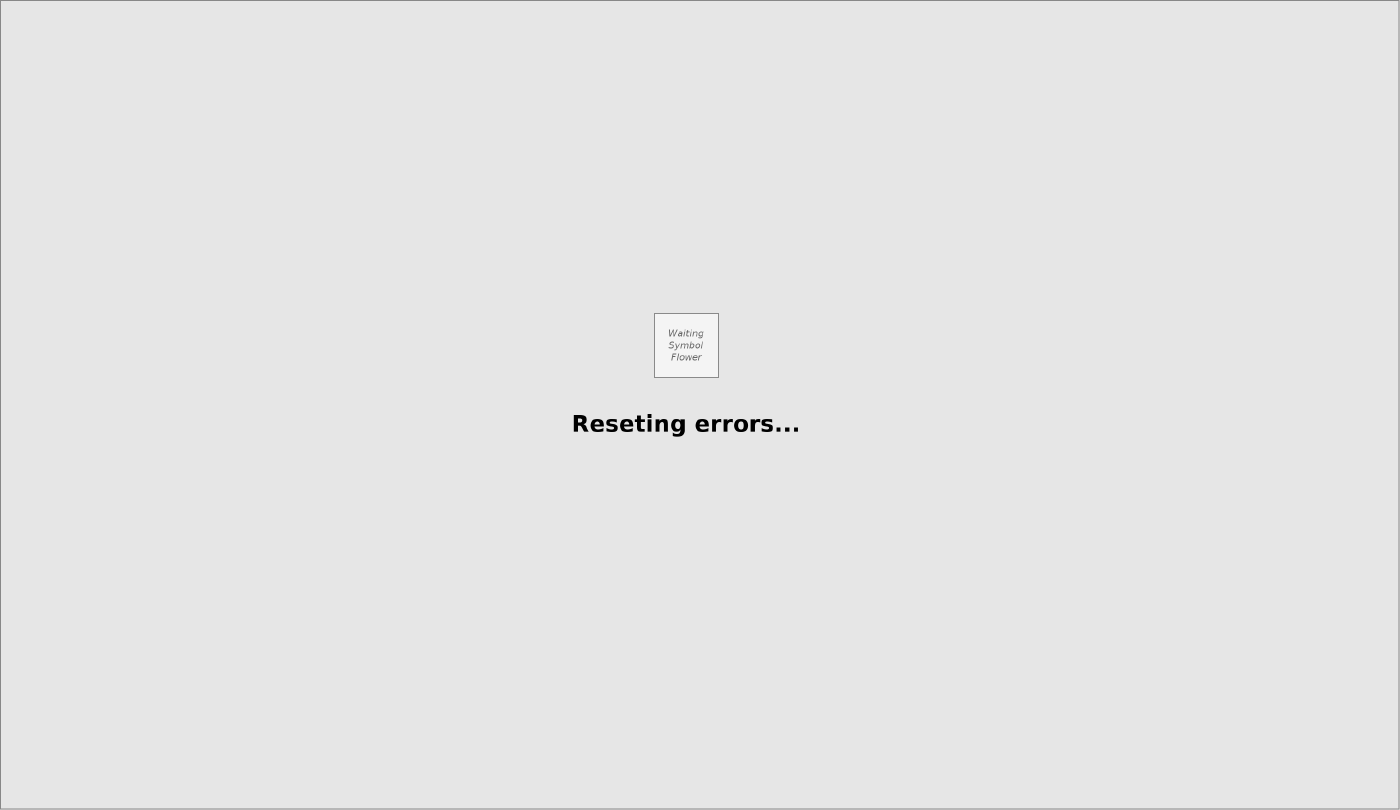
VISUALIZATION PageReset  // 1520x880
    WaitingSymbolFlower (710,340 70x70)
    Label (570,440 350x40), "Reseting errors..."
END_VISUALIZATION

(* stored: Version 1.1.0.1, ProductVersion 3.1.4024.9
   Visu PageReset: Id {255dff00-129e-4f3a-988a-71d6e5880867} *)
